(* PLC project Generated.project, CODESYS CODESYS V3.5 SP19 Patch 1 *)
(* stored: creationDateTime 2026-09-03T14:37:01.782708, modificationDateTime 2026-09-03T14:37:01.782708 *)

(* ═══════════════════════════════════════════════════════════════ 🎯 ST_MachineHomingHMI — Données d'échange IHM du cycle de référencement machine ─────────────────────────────────────────────────────────────── 📄 Structuration Cmd / State / Cfg , homogène avec ST_CycleHMI / ST_CycleDiveSearchHMI / ST_CycleExtractionHMI. ═══════════════════════════════════════════════════════════════ *)
TYPE ST_MachineHomingHMI : STRUCT
  Cmd : ST_MachineHomingCmd;
  State : ST_MachineHoming;  (* Image publiée du FB_MachineHomingCycle (SeqStep, Step, Instruction, Failed, ordres, …) *)
  Cfg : ST_MachineHomingCfg;
END_STRUCT;
END_TYPE

(* ======================================================================= 🧭 ST_MachineHoming — Etat publie du homing conjoint machine (M1/M2/benne) ─────────────────────────────────────────────────────────────── 🎯 Rôle : Regroupe les 8 sorties homing a plat de PRG_02_Acquisition en un bus struct unique, publie sur le bus inter-PRG. 🔒 Sécurité : Homed = qualification conjointe reference machine (gate SEMI_AUTO). HomingLoss = perte reference en mouvement : arret controle SafeStop. 📄 Doc métier : DOC/AF/AF_Partie-09_Fonction_Encoder_v2.4.md (F09.08) ======================================================================= *)
TYPE ST_MachineHoming : STRUCT
  Homed : BOOL;  (* Qualification conjointe reference machine *)
  SetPosBucketOpen : BOOL;  (* Valider position actuelle = reference benne ouverte *)
  SetPosBucketClose : BOOL;  (* Valider position actuelle = reference benne fermee *)
  Active : BOOL;  (* Homing conjoint en cours *)
  HomingLoss : BOOL;  (* Perte reference en mouvement : arret controle SafeStop *)
  Step : INT;  (* Etape guidee reference (echelle de priorite E_MachineHomingStep) *)
  Instruction : STRING(120);  (* Consigne IHM reference *)
  Failed : BOOL;  (* Transaction reference abandonnee *)
  SeqStep : INT;  (* Step GRAFCET courant (E_MachineHomingTxState HX0..HXF) *)
  M3Locked : BOOL;  (* Translation M3 interdite pendant le cycle de homing machine *)
  CmdWinchM1 : ST_ProgramWinchRequest;  (* Ordre treuil M1 couple palier 1 (HX2 montee / HX3 descente) *)
  CmdWinchM2 : ST_ProgramWinchRequest;  (* Ordre treuil M2 couple palier 1 (HX2 montee / HX3 descente) *)
  CmdBucketOpen : BOOL;  (* Ordre ouverture benne palier 1 sans FDC soft (HX4) *)
  CmdBucketClose : BOOL;  (* Ordre fermeture benne palier 1 sans FDC soft (HX4) *)
END_STRUCT;
END_TYPE

(* ═══════════════════════════════════════════════════════════════ ⚙️ ST_MachineHomingCfg — Réglages IHM du cycle de référencement machine ─────────────────────────────────────────────────────────────── 🎯 Mise en service. Les réglages géométriques (positions capteur, offsets benne) restent portés par GVL_PERSISTENT (_WinchM1CfgPersist / _BucketCfgPersist). 💾 Ponté vers persist (_MachineHomingCfgPersist) via FB_CfgPersistBridge_MachineHomingCfg. ═══════════════════════════════════════════════════════════════ *)
TYPE ST_MachineHomingCfg : STRUCT
  ForceStepTarget : INT := 0;  (* 🔧 Step GRAFCET cible du forçage (0=HX0 .. 9=HXF), borné côté FB *)
  Initialized : BOOL := FALSE;  (* 🚦 flag restauration boot *)
END_STRUCT;
END_TYPE

(* ═══════════════════════════════════════════════════════════════ 🎮 ST_MachineHomingCmd — Commandes IHM du cycle de référencement machine ─────────────────────────────────────────────────────────────── 🎯 Cycle homing machine (FB_MachineHomingCycle) — orchestré en MAINT_N2. Séparé de ST_CycleCmd (cycle SEMI_AUTO) et de ST_ModesCmd (modes de marche). Boutons momentanés uniquement ; réglages -> ST_MachineHomingCfg. ═══════════════════════════════════════════════════════════════ *)
TYPE ST_MachineHomingCmd : STRUCT
  BtnStart : BOOL;  (* ▶️ Lancer le cycle de homing machine (MAINT_N2, front) — alternative au motif 3 appuis joystick *)
  BtnValidate : BOOL;  (* ✅ Validation depuis IHM (front) — équivaut à 1 appui du motif 3 appuis joystick *)
  BtnAbort : BOOL;  (* ⏹️ Quitter / abandonner le cycle homing (front) — retour HX0 sans mouvement *)
  TglCommissioning : BOOL := FALSE;  (* 🔧 Case mise en service : déverrouille le forçage de step (MAINT_N2). NON persisté (reset au reboot = sûr). *)
  BtnForceStepApply : BOOL;  (* 🔧 Applique le forçage de step (front) — impulsion ; cible = ST_MachineHomingCfg.ForceStepTarget *)
END_STRUCT;
END_TYPE

(* ======================================================================= 🔌 ST_ProgramWinchRequest — Demande de mouvement treuil par le programme ─────────────────────────────────────────────────────────────── 🎯 Rôle : Regroupe les demandes logiques de treuil formulées par le séquenceur 📄 Référentiel : DOC/WFLOW/CONTRACTS/INTERPRG_CONTRACT_PRG03_MODES_CYCLE_v1.0.md ======================================================================= *)
TYPE ST_ProgramWinchRequest : STRUCT
  RunRequest : BOOL;  (* Ordre marche demandé par le programme *)
  ReqAscent : BOOL;  (* Demande montée *)
  ReqDescend : BOOL;  (* Demande descente *)
  StepTgt : INT;  (* Palier de vitesse cible demandé (1 à 5, 0 = arrêt) *)
END_STRUCT;
END_TYPE
